TYPE ST_MainCabinet_HWQ :
STRUCT
  //outputs
  bEmgyBtnWhiteLight  	: BOOL;  
  bEmgyBtnRedLight  		: BOOL; 
  
  stStackLight          : ST_StackLight_HWQ;
END_STRUCT
END_TYPE

(* stored: Version 1.1.0.1, ProductVersion 3.1.4024.12
   DUT ST_MainCabinet_HWQ: Id {fa88e60a-08e3-4b56-84c0-1ff06fc8ebb1} *)
